// TwinCAT 3 PLC project Tolerantie_waardes
// ProgramVersion: 3.1.4024.0
// libraries:
//   Tc2_Standard, * (Beckhoff Automation GmbH)
//   Tc2_System, * (Beckhoff Automation GmbH)
//   Tc3_Module, * (Beckhoff Automation GmbH)
// project tree:
//   / PlcTask.TcTTO
//   POUs/ MAIN.TcPOU
// (motion and I/O tree: see PLC project potentiometer_inlezen)
// real-time tasks:
//   TASK PlcTask: cycle T#10ms, priority 20, ADS port 350
//   TASK PlcTask1: cycle T#10ms, priority 21, ADS port 351
//   TASK PlcTask2: cycle T#10ms, priority 22, ADS port 352
//   TASK PlcTask3: cycle T#10ms, priority 26, ADS port 353
//   TASK PlcTask4: cycle T#10ms, priority 25, ADS port 354
//   TASK PlcTask5: cycle T#10ms, priority 24, ADS port 355
//   TASK PlcTask6: cycle T#10ms, priority 23, ADS port 356
//   TASK PlcTask7: cycle T#10ms, priority 27, ADS port 357

CONFIGURATION Tolerantie_waardes
    RESOURCE PLC ON TwinCAT3
        TASK PlcTask(INTERVAL := T#10ms, PRIORITY := 23);
        PROGRAM MAIN WITH PlcTask : MAIN;
    END_RESOURCE
END_CONFIGURATION

// ---- POUs/MAIN.TcPOU
PROGRAM MAIN
VAR
	
// Inputs
	nGemeten AT %I*: REAL; // Fysieke potentiometer 
	nGevraagd     : INT; // gevraagde waarde ( Visualisatie)
	
// Outputs
	groeneLamp    AT %Q*:BOOL;
	rodeLamp      AT %Q*:BOOL;
	
END_VAR

(*
Tolerantiewaardes (2 regels)

Lees een fysieke potentiometer in als de variabele nGemeten en een potiometer via de visualisatie in als nGevraagd. 

Als de gemeten waarde kleiner is dan de gewenste waarde met een tolerantie van 10%, dan moet de rode lamp branden. 

Als de gemeten waarde groter is dan de gewenste waarde met een tolerantie van 10%, dan moet de groene lamp branden.
*)

rodeLamp	:=(nGevraagd-(10*(nGevraagd/100))) > (100*nGemeten/32767); // Berekend waarde 10% minder THEN gevraagde waarde -> LAMP AAN
groeneLamp	:=(nGevraagd+(10*(nGevraagd/100))) < (100*nGemeten/32767); // Berekend waarde 10% meer   THEN gevraagde waarde -> LAMP AAN

END_PROGRAM
